FUNCTION_BLOCK InputCompressor (* Basic Function Block Type *)
  (* Standard: 61499-2 *)
  (* Version 0.0, 6/21/2018, Rediska, nxtControl GmbH, Template *)
  PACKAGE Main;
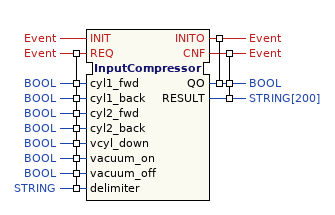
  EVENT_INPUT
    INIT; (* Initialization Request *)
    REQ WITH cyl1_fwd, cyl1_back, cyl2_fwd, cyl2_back, vcyl_down, vacuum_on, vacuum_off, delimiter; (* Normal Execution Request *)
  END_EVENT
  EVENT_OUTPUT
    INITO WITH QO; (* Initialization Confirm *)
    CNF WITH QO, RESULT; (* Execution Confirmation *)
  END_EVENT
  VAR_INPUT
    cyl1_fwd : BOOL;
    cyl1_back : BOOL;
    cyl2_fwd : BOOL;
    cyl2_back : BOOL;
    vcyl_down : BOOL;
    vacuum_on : BOOL;
    vacuum_off : BOOL;
    delimiter : STRING;
  END_VAR
  VAR_OUTPUT
    QO : BOOL; (* Output event qualifier *)
    RESULT : STRING[200];
  END_VAR
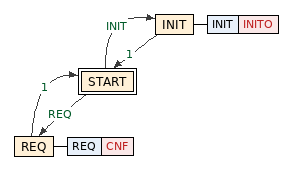
  EC_STATES
    START; (* Initial State *)
    INIT : INIT -> INITO; (* Initialization *)
    REQ : REQ -> CNF; (* Normal execution *)
  END_STATES
  EC_TRANSITIONS
    START TO INIT := INIT;
    INIT TO START := 1;
    START TO REQ := REQ;
    REQ TO START := 1;
  END_TRANSITIONS
  ALGORITHM INIT IN ST: (* Initialization algorithm *)
QO:=TRUE;
  END_ALGORITHM
  ALGORITHM REQ IN ST: (* Normally executed algorithm *)
RESULT :=
CONCAT(
  CONCAT(
    BOOL_TO_STRING(cyl1_fwd), delimiter,
    BOOL_TO_STRING(cyl1_back), delimiter,
    BOOL_TO_STRING(cyl2_fwd), delimiter
  ),
  CONCAT(
    BOOL_TO_STRING(cyl2_back), delimiter,
    BOOL_TO_STRING(vcyl_down), delimiter,
    BOOL_TO_STRING(vacuum_on), delimiter,
    BOOL_TO_STRING(vacuum_off), delimiter
  ),
  "$N");
  END_ALGORITHM
END_FUNCTION_BLOCK
